{attribute 'GeneratedUsingTerminal: EL5101-0011-0016'}
{attribute addProperty BoxType "EL5101-0011-0016"}
{attribute addProperty Id "ARRAY_0UDINT4"}
{attribute addProperty CRC "3791446571"}
{attribute addProperty Size "4"}
TYPE Counter_value_E1FCE22B :
STRUCT
	{attribute addProperty Name "ARRAY_0"}
	ARRAY_0 : UDINT;
END_STRUCT
END_TYPE

(* stored: Version 1.2.0.0, ProductVersion 3.1.4024.9
   DUT Counter_value_E1FCE22B: Id {6dfa117a-bcb0-4fae-b952-19a51e46a808} *)
